# B&R Automation Studio project TrakDemo (part 2)

#### Cyclic.st - Cyclic code
```iecst
PROGRAM _CYCLIC
	(* catch shuttle on gSegB7 for simulation of shuttle errors *)
	fbCatchShuttle();

	(* assembly's state machine *)
	fbLogStep.EventID := TRAK_BASIC_INFO_ID;

	CASE step OF
		ASM_INIT:
		fbGetInfo( Execute := FALSE ); (* reset fb *)
		fbGetInfo( Execute := TRUE );
		fbPowerOn( Execute := FALSE ); (* reset fb *)
		fbPowerOff( Execute := FALSE ); (* reset fb *)
		step := ASM_GET_INFO;

		ASM_GET_INFO:
		fbLogStep.Signal := 'ASM_GET_INFO';
		IF fbGetInfo.Done THEN
			fbGetInfo( Execute := FALSE ); (* reset fb *)
			assemblyCtrl.Status.SimulationOnPlcMode := fbGetInfo.AssemblyInfo.SimulationOnPlcMode;
			step := ASM_W_READY_FOR_POWER_ON;
		ELSIF fbGetInfo.Error THEN
			fbGetInfo( Execute := FALSE ); (* reset fb *)
			step := ASM_ERR_GET_INFO;
			fbLogStep.EventID := TRAK_BASIC_ERROR_ID;
			fbLogStep.Signal := 'ASM_ERR_GET_INFO';
		ELSE (* busy *)
			fbGetInfo();
		END_IF

		ASM_W_READY_FOR_POWER_ON:
		fbLogStep.Signal := 'ASM_W_READY_FOR_POWER_ON';
		IF assemblyCtrl.Status.Info.ReadyForPowerOn THEN
			IF assemblyCtrl.Status.Info.PowerOn THEN
				step := ASM_POWER_IS_ON;
			ELSE
				step := ASM_POWER_IS_OFF;
			END_IF
		END_IF

		ASM_POWER_IS_OFF:
		fbLogStep.Signal := 'ASM_POWER_IS_OFF';
		IF assemblyCtrl.Cmd.PowerOn THEN
			assemblyCtrl.Cmd.PowerOn := FALSE;
			fbPowerOn( Execute := TRUE );
			step := ASM_W_POWER_ON;
		END_IF

		ASM_ADD_SIM_SHUTTLES:
		fbLogStep.Signal := 'ASM_ADD_SIM_SHUTTLES';
		IF fbAddSimShuttle.Done THEN
			fbAddSimShuttle( Execute := FALSE ); (* reset fb *)
			IF assemblyCtrl.Status.Info.ShuttlesCount >= assemblyCtrl.Para.NumberOfSimulatedShuttles OR assemblyCtrl.Para.NumberOfSimulatedShuttles = 0 THEN
				step := ASM_POWER_IS_ON;
			ELSE
				fbAddSimShuttle.Position := fbAddSimShuttle.Position + 0.06;
				fbAddSimShuttle( Execute := TRUE );
			END_IF
		ELSIF fbAddSimShuttle.Error THEN
			fbAddSimShuttle( Execute := FALSE ); (* reset fb *)
			step := ASM_ERR_ADDING_SHUTTLE;
			fbLogStep.EventID := TRAK_BASIC_ERROR_ID;
			fbLogStep.Signal := 'ASM_ERR_ADDING_SHUTTLE';
		ELSE (* busy *)
			fbAddSimShuttle();
		END_IF

		ASM_W_POWER_ON:
		fbLogStep.Signal := 'ASM_W_POWER_ON';
		IF fbPowerOn.Done AND assemblyCtrl.Status.Info.PowerOn THEN
			fbPowerOn( Execute := FALSE );  (* reset fb *)
			IF assemblyCtrl.Status.Info.ShuttlesCount >= assemblyCtrl.Para.NumberOfSimulatedShuttles THEN
				step := ASM_POWER_IS_ON;
			ELSE
				fbAddSimShuttle( Execute := FALSE ); (* reset fb *)
				fbAddSimShuttle( Execute := TRUE );
				step := ASM_ADD_SIM_SHUTTLES;
			END_IF
		ELSIF fbPowerOn.Error THEN
			fbPowerOn( Execute := FALSE );  (* reset fb *)
			step := ASM_ERR_POWERING_ON;
			fbLogStep.EventID := TRAK_BASIC_ERROR_ID;
			fbLogStep.Signal := 'ASM_ERR_POWERING_ON';
		ELSE (* busy *)
			fbPowerOn();
		END_IF

		ASM_POWER_IS_ON:
		fbLogStep.Signal := 'ASM_POWER_IS_ON';
		IF NOT assemblyCtrl.Status.Info.PowerOn THEN
			step := ASM_POWER_IS_OFF;
		ELSIF assemblyCtrl.Cmd.PowerOff THEN
			assemblyCtrl.Cmd.PowerOff := FALSE;
			fbPowerOff( Execute := TRUE );
			step := ASM_W_POWER_OFF;
		ELSIF assemblyCtrl.Cmd.Start THEN
			assemblyCtrl.Cmd.Start := FALSE;
			fbStartShuttles( Execute := FALSE ); (* reset fb *)
			fbStartShuttles( Execute := TRUE ); (* reset fb *)
			step := ASM_START_MOVEMENT;
		ELSIF assemblyCtrl.Cmd.SimSegmentError THEN
			assemblyCtrl.Cmd.SimSegmentError := FALSE;
			fbSegCommandError( Segment := ADR(gSegB7), Type := TD_SEGERRCMD_SEGMENT, Execute := FALSE ); (* reset fb *)
			fbSegCommandError( Execute := TRUE );
			step := ASM_SIMULATE_ERROR;
		ELSIF assemblyCtrl.Cmd.SimChannelError THEN
			IF assemblyCtrl.Status.AllShuttlesMoving THEN
				assemblyCtrl.Cmd.SimChannelError := FALSE;
				fbSegCommandError( Segment := ADR(gSegB7), Type := TD_SEGERRCMD_CHANNEL, Execute := FALSE ); (* reset fb *)
				shuttleCounter := fbCatchShuttle.ShuttleCounter;
				step := ASM_WAIT_FOR_DEFECT_SHUTTLE;
			ELSE
				assemblyCtrl.Cmd.SimChannelError := FALSE;
			END_IF
		ELSIF assemblyCtrl.Cmd.SimEncoderError  THEN
			IF assemblyCtrl.Status.AllShuttlesMoving THEN
				assemblyCtrl.Cmd.SimEncoderError := FALSE;
				fbSegCommandError( Segment := ADR(gSegB7), Type := TD_SEGERRCMD_ENCODER, Execute := FALSE ); (* reset fb *)
				shuttleCounter := fbCatchShuttle.ShuttleCounter;
				step := ASM_WAIT_FOR_DEFECT_SHUTTLE;
			ELSE
				assemblyCtrl.Cmd.SimEncoderError := FALSE;
			END_IF
		END_IF

		ASM_START_MOVEMENT:
		fbLogStep.Signal := 'ASM_START_MOVEMENT';
		IF fbStartShuttles.Done THEN
			fbStartShuttles( Execute := FALSE ); (* reset fb *)
			step := ASM_POWER_IS_ON;
		ELSIF fbStartShuttles.Error THEN
			fbStartShuttles( Execute := FALSE ); (* reset fb *)
			step := ASM_ERR_START_MOVEMENT;
			fbLogStep.EventID := TRAK_BASIC_ERROR_ID;
			fbLogStep.Signal := 'ASM_ERR_START_MOVEMENT';
		ELSE (* busy *)
			fbStartShuttles();
		END_IF

		ASM_SIMULATE_ERROR:
		fbLogStep.Signal := 'ASM_SIMULATE_ERROR';
		IF fbSegCommandError.Done THEN
			fbSegCommandError( Execute := FALSE );
			step := ASM_POWER_IS_ON;
		ELSIF fbSegCommandError.Error THEN
			fbSegCommandError( Execute := FALSE );
			step := ASM_POWER_IS_ON;
//			step := ASM_ERR_SIMULATE_ERROR;
//			fbLogStep.EventID := TRAK_BASIC_ERROR_ID;
//			fbLogStep.Signal := 'ASM_ERR_SIMULATE_ERROR';
		ELSE (* busy *)
			fbSegCommandError();
		END_IF

		ASM_WAIT_FOR_DEFECT_SHUTTLE: (* wait for defect shuttle passing *)
		fbLogStep.Signal := 'ASM_WAIT_FOR_DEFECT_SHUTTLE';
		IF shuttleCounter <> fbCatchShuttle.ShuttleCounter THEN
			fbSegCommandError( Execute := TRUE );
			assemblyCtrl.Cmd.SimChannelError := FALSE;
			assemblyCtrl.Cmd.SimEncoderError := FALSE;
			step := ASM_SIMULATE_ERROR;
		END_IF

		ASM_W_POWER_OFF:
		fbLogStep.Signal := 'ASM_W_POWER_OFF';
		IF fbPowerOff.Done OR  NOT assemblyCtrl.Status.Info.PowerOn THEN
			step := ASM_POWER_IS_OFF;
			fbPowerOff( Execute := FALSE ); (* reset fb *)
		ELSIF fbPowerOff.Error THEN
			fbPowerOff( Execute := FALSE ); (* reset fb *)
			step := ASM_ERR_POWERING_OFF;
			fbLogStep.EventID := TRAK_BASIC_ERROR_ID;
			fbLogStep.Signal := 'ASM_ERR_POWERING_OFF';
		ELSE (* busy *)
			fbPowerOff();
		END_IF

		ASM_ERR_GET_INFO..ASM_ERR_GENERAL:

	END_CASE

	assemblyCtrl.Status.Step := step;
	fbLogStep(); (* log state machine *)

	(* read assembly status *)
	fbReadStatus();
	assemblyCtrl.Status.Disabled  	:= fbReadStatus.AssemblyDisabled;
	assemblyCtrl.Status.ErrorStop 	:= fbReadStatus.AssemblyErrorStop;
	assemblyCtrl.Status.Homing 		:= fbReadStatus.AssemblyHoming;
	assemblyCtrl.Status.Stopping 	:= fbReadStatus.AssemblyStopping;
	assemblyCtrl.Status.Ready 	  	:= fbReadStatus.AssemblyReady;

	(* read assembly info *)
	fbReadInfo();
	assemblyCtrl.Status.Info := fbReadInfo.AssemblyInfo;
	assemblyCtrl.Status.AllShuttlesMoving := FALSE;
	IF assemblyCtrl.Status.Info.ShuttlesCount = assemblyCtrl.Para.NumberOfSimulatedShuttles THEN
		IF assemblyCtrl.Status.Info.ShuttlesInDisabledCount = 0 AND
			assemblyCtrl.Status.Info.ShuttlesInErrorStopCount = 0 AND
			assemblyCtrl.Status.Info.ShuttlesInStandstillCount = 0 AND
			assemblyCtrl.Status.Info.ShuttlesInStoppingCount = 0 THEN
			assemblyCtrl.Status.AllShuttlesMoving := TRUE;
		END_IF
	END_IF

	(* run recorder for breakdown analysis *)
	fbRecorder(Trigger := assemblyCtrl.Status.ErrorStop );
	(* web page *)
	fbWebServices();

	(* reset error stop *)
	fbLogResetStep.EventID := TRAK_BASIC_INFO_ID;
	CASE assemblyCtrl.Status.ResetStep OF
		ASMR_NO_ERROR:
		fbLogResetStep.Signal := 'ASMR_NO_ERROR';
		IF assemblyCtrl.Status.ErrorStop THEN
			fbAsmReset( Execute := FALSE ); (* reset fb *)
			assemblyCtrl.Cmd.Reset := FALSE;
			assemblyCtrl.Status.ResetStep := ASMR_W_ACKNOWLEDGE;
		END_IF

		ASMR_W_ACKNOWLEDGE:
		fbLogResetStep.Signal := 'ASMR_W_ACKNOWLEDGE';
		IF assemblyCtrl.Cmd.Reset THEN
			assemblyCtrl.Cmd.Reset := FALSE;
			fbAsmReset( Execute := TRUE ); (* reset fb *)
			assemblyCtrl.Status.ResetStep := ASMR_RESET;
		END_IF

		ASMR_RESET:
		fbLogResetStep.Signal := 'ASMR_RESET';
		IF fbAsmReset.Done THEN
			fbAsmReset( Execute := FALSE ); (* reset fb *)
			assemblyCtrl.Status.ResetStep := ASMR_NO_ERROR;
		ELSIF fbAsmReset.Error THEN
			fbAsmReset( Execute := FALSE ); (* reset fb *)
			assemblyCtrl.Status.ResetStep := ASMR_INTERNAL_ERROR;
			fbLogResetStep.EventID := TRAK_BASIC_ERROR_ID;
			fbLogResetStep.Signal := 'ASMR_INERNAL_ERROR';
		ELSE (* busy *)
			fbAsmReset();
		END_IF

		ASMR_INTERNAL_ERROR:

	END_CASE

	fbLogResetStep(); (* log state machine *)

END_PROGRAM
```

#### Init.st - Init code
```iecst
PROGRAM _INIT
	gSecOvalA;
	gSecOvalB;
	gSecCompleteLoop;

	fbReadStatus.Assembly := ADR(gAssembly_1);
	fbReadStatus.Enable := TRUE;

	fbReadInfo.Assembly := fbReadStatus.Assembly;
	fbReadInfo.Enable := TRUE;

	fbGetInfo.Assembly := fbReadStatus.Assembly;

	fbPowerOn.Assembly := fbReadStatus.Assembly;

	fbPowerOff.Assembly := fbReadStatus.Assembly;

	fbStartShuttles.Sector := gSecCompleteLoop;
	fbStartShuttles.TargetSector := gSecCompleteLoop;
	fbStartShuttles.Acceleration := 4.0;
	fbStartShuttles.Deceleration := 4.0;
	fbStartShuttles.Velocity := 2.0;
	fbStartShuttles.Jerk := 0.0;
	fbStartShuttles.Direction := mcDIR_POSITIVE;

	fbAddSimShuttle.Sector := ADR(gSecCompleteLoop);
	fbAddSimShuttle.Position := 0.5;

	fbAddSimShuttle.AdvancedParameters.Velocity := 0.0;
	fbAddSimShuttle.AdvancedParameters.Orientation := mcDIR_POSITIVE;
	fbAddSimShuttle.AdvancedParameters.Deceleration := 6.0;
	fbAddSimShuttle.AdvancedParameters.Virtual := FALSE;

	fbCatchShuttle.ProcessPoint := PP_ErrorPosition1;
	fbCatchShuttle.Enable := TRUE;

	fbAsmReset.Assembly := ADR(gAssembly_1);

	fbRecorder.AssemblyName := 'gAssembly_1';
	fbRecorder.FileDeviceName := 'Diagnosis';
	fbRecorder.FileNamePrefix := 'Demo_';
	fbRecorder.MaxNumberOfRecordings := 10;
	fbRecorder.DataAddress := ADR(shuttleData);
	fbRecorder.DataSize := SIZEOF(shuttleData); (* type of McAcpTrakShuttleData[] if no shuttle user data is defined, see MC_BR_AsmCopyShuttleData_AcpTrak *)
	fbRecorder.UserDataSize := 0;
	fbRecorder.Enable := TRUE;

	fbWebServices.AssemblyName := fbRecorder.AssemblyName;
	fbWebServices.DataAddress := fbRecorder.DataAddress;
	fbWebServices.DataSize := fbRecorder.DataSize;
	fbWebServices.UserDataSize := fbRecorder.UserDataSize;
	fbWebServices.Enable := TRUE;

	assemblyCtrl.Para.NumberOfSimulatedShuttles := 10;
	assemblyCtrl.SizeOf := SIZEOF(assemblyCtrl);

	step := ASM_INIT;

	fbLogStep( Enable := FALSE, LogName := 'MyTrak', SignalName := 'AssCtrl Step', EventID := TRAK_BASIC_INFO_ID );
	fbLogStep.Enable := TRUE;

	fbLogResetStep( Enable := FALSE, LogName := 'MyTrak', SignalName := 'AssCtrl ResetStep', EventID := TRAK_BASIC_INFO_ID );
	fbLogResetStep.Enable := TRUE;
END_PROGRAM
```

#### Variables.var - Local variables
```iecst
VAR
	fbStartShuttles : TL_StartShuttlesInSector;
	fbLogResetStep : TD_LogWatchSTRING;
	fbLogStep : TD_LogWatchSTRING;
	fbAddSimShuttle : MC_BR_SecAddShuttle_AcpTrak;
	fbPowerOff : MC_BR_AsmPowerOff_AcpTrak;
	fbPowerOn : MC_BR_AsmPowerOn_AcpTrak;
	fbGetInfo : MC_BR_AsmGetInfo_AcpTrak;
	fbReadInfo : MC_BR_AsmReadInfo_AcpTrak;
	fbReadStatus : MC_BR_AsmReadStatus_AcpTrak;
	fbWebServices : TD_WebServices;
	fbCatchShuttle : TL_CatchShuttle;
	fbRecorder : TD_Recorder;
	step : AssemblyStepEnum;
	fbAsmReset : MC_BR_AsmReset_AcpTrak;
	fbSegCommandError : TD_SegCommandError;
	assemblyCtrl : AssemblyType;
	shuttleData : ARRAY[0..49] OF McAcpTrakShuttleData;
	shuttleCounter : DINT;
END_VAR
```

Listed in the project but not available here: Logical/Global.typ, Logical/Global.var, Logical/Trak/AssCtrl1/Exit.st, Logical/Trak/AssCtrl2/Exit.st, Logical/Trak/AssCtrl/Exit.st
